FUNCTION_BLOCK AnalogInput_Status_HMI (* Service Interface Function Block Type *)
  (* Standard: 61499-2 *)
  (* Version 0.0, 8/31/2022, SESA583220, Schneider Electric, template *)
  PACKAGE SE.Nereda;
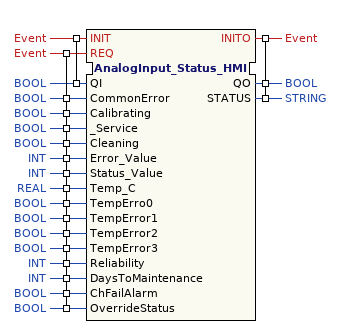
  EVENT_INPUT
    INIT WITH QI;
    REQ WITH CommonError, Calibrating, _Service, Cleaning, Error_Value, Status_Value, Temp_C, TempErro0, TempError1, TempError2, TempError3, Reliability, DaysToMaintenance, ChFailAlarm, OverrideStatus;
  END_EVENT
  EVENT_OUTPUT
    INITO WITH QO, STATUS;
  END_EVENT
  VAR_INPUT
    QI : BOOL;
    CommonError : BOOL;
    Calibrating : BOOL;
    _Service : BOOL;
    Cleaning : BOOL;
    Error_Value : INT;
    Status_Value : INT;
    Temp_C : REAL;
    TempErro0 : BOOL;
    TempError1 : BOOL;
    TempError2 : BOOL;
    TempError3 : BOOL;
    Reliability : INT;
    DaysToMaintenance : INT;
    ChFailAlarm : BOOL;
    OverrideStatus : BOOL;
  END_VAR
  VAR_OUTPUT
    QO : BOOL; (* Event Output Qualifier *)
    STATUS : STRING; (* Service Status *)
  END_VAR
  SERVICE /
    SEQUENCE 
    END_SEQUENCE
  END_SERVICE
END_FUNCTION_BLOCK
